INTERFACE ITF_MCMachineControl_HMI_Init EXTENDS ITF_BaseTopElement, ITF_MCMachineControl_HMI_Connector

END_INTERFACE

(* stored: Version 1.1.0.1
   Itf ITF_MCMachineControl_HMI_Init: Id {3cb73cc3-b9bc-03be-306b-d8030f881dde} *)
